KUKA KRL program: HOME.src, home.dat

--- HOME.src ---
&ACCESS RVO1
&REL 5
&COMMENT 03-10-R1 MOVE HOME
&PARAM EDITMASK = *
DEF HOME( )
;FOLD INI
  ;FOLD BASISTECH INI
    GLOBAL INTERRUPT DECL 3 WHEN $STOPMESS==TRUE DO IR_STOPM ( )
    INTERRUPT ON 3
    BAS (#INITMOV,0 )
  ;ENDFOLD (BASISTECH INI)
  ;FOLD USER INI
    ;Make your modifications here

  ;ENDFOLD (USER INI)
;ENDFOLD (INI)
;********************************
; Gestamp Standards
; Line - BMW G65 (cell 03)
; Robot 03-10-R1 (BMW-03-10-R1)
; Application - MOVE HOME
;********************************
; DIRECT PTP MOVE TO HOME FROM THE CURRENT POSITION - NO VIA POINTS. P1 (home.dat) HAS THE
; SAME AXIS VALUES AS XHOME ($config.dat); THE FORM IS A KSS 4.1.5 ONE (OLD BAS CALLS)
;********************************
;NOTE: THE ONLY CALLER IS CELL, AFTER InitializeSystem, WHOSE HomeCheck HAS ALREADY BROUGHT
;NOTE: THE ROBOT INTO THE HOME WINDOW ($IN_HOME)
;FOLD PTP P1 Vel=100 % PDAT1 Tool[1]:TOOL 1 Base[0];%{PE}%R 4.1.5,%MKUKATPBASIS,%CMOVE,%VPTP,%P 1:PTP, 2:P1, 3:, 5:100, 7:PDAT1
$BWDSTART=FALSE
PDAT_ACT=PPDAT1
BAS(#PTP_DAT)
FDAT_ACT=FP1
BAS(#FRAMES)
BAS(#VEL_PTP,100)
PTP XP1
;ENDFOLD
END

--- home.dat ---
&ACCESS RVO1
&REL 5
&PARAM EDITMASK = *
DEFDAT  home
;FOLD EXTERNAL DECLARATIONS;%{PE}%MKUKATPBASIS,%CEXT,%VCOMMON,%P
;FOLD BASISTECH EXT;%{PE}%MKUKATPBASIS,%CEXT,%VEXT,%P
EXT  BAS (BAS_COMMAND  :IN,REAL  :IN )
DECL INT SUCCESS
;ENDFOLD (BASISTECH EXT)
;FOLD USER EXT;%{E}%MKUKATPUSER,%CEXT,%VEXT,%P
;Make here your modifications

;ENDFOLD (USER EXT)
;ENDFOLD (EXTERNAL DECLARATIONS)
DECL E6AXIS XP1={A1 11.0530167,A2 -136.848862,A3 85.1306381,A4 -8.17127800,A5 54.4414291,A6 184.387085,E1 0.0,E2 0.0,E3 0.0,E4 0.0,E5 0.0,E6 0.0}
DECL FDAT FP1={TOOL_NO 1,BASE_NO 0,IPO_FRAME #BASE}
DECL PDAT PPDAT1={VEL 100.000,ACC 100.000,APO_DIST 0.0}
ENDDAT
